// TIA Portal V18 export
FUNCTION_BLOCK "manual_analog"   // FB7, FBD
{ S7_Optimized_Access := 'TRUE' }
VERSION : 0.1
// stored: AutoNumber true, IsIECCheckEnabled false, IsRetainMemResEnabled false, MemoryReserve 100, SetENOAutomatically false, UDAEnableTagReadback false
   VAR_INPUT
      ALLOWED : Bool;
      ALLOWED_ONLY_IN_OVERRIDE : Bool;
      OVERRIDE_NOW : Bool;
      isMultiturn : Bool;
      POS : Real;
      SET_SPEED : Real;
      xFwdOk : Bool;
      xRevOk : Bool;
      clibrated : Bool;
      par_spd_absmax : Real := 1000.0;
      par_dist_absmax : Real := 100.0;
      par_speed_crawl : Real;
      par_dist_crawl : Real;
      par_dist_stop : Real := 10.0;
      par_spd_blind : Real := 500.0;
      par_fwd_limit : Real := 10000.0;
      par_rev_limit : Real := 0.0;
      par_t_acc : Real;
   END_VAR
   VAR_OUTPUT
      SPEED : Real;
      ER_settings : Bool;
      er_ws : WString;
   END_VAR
   VAR
      speed_slowly_accelerated : Real;
      mot_speed_wdir_slowly_accelerated_Instance { S7_SetPoint := 'True'} : "mot_speed_wdir_slowly_accelerated";
   END_VAR
   VAR_TEMP
      speed_calculated : Real;
      speed_calc_abs : Real;
      estop_ok_no_err : Bool;
      blind : Bool;
      set_spd_loc : Real;
   END_VAR
   VAR CONSTANT
      erwsnoer : WString := WSTRING#'no er';
      erws1 : WString := WSTRING#'lim fwd = rev';
      erws2 : WString := WSTRING#'#par_dist_fast 0';
      erws3 : WString := WSTRING#'#par_spd_absmax';
   END_VAR
   VAR_TEMP   // added for the SCL form of the ladder/FBD networks
      _w1 : Bool;
      _w2 : Bool;
   END_VAR
BEGIN

REGION Network 1
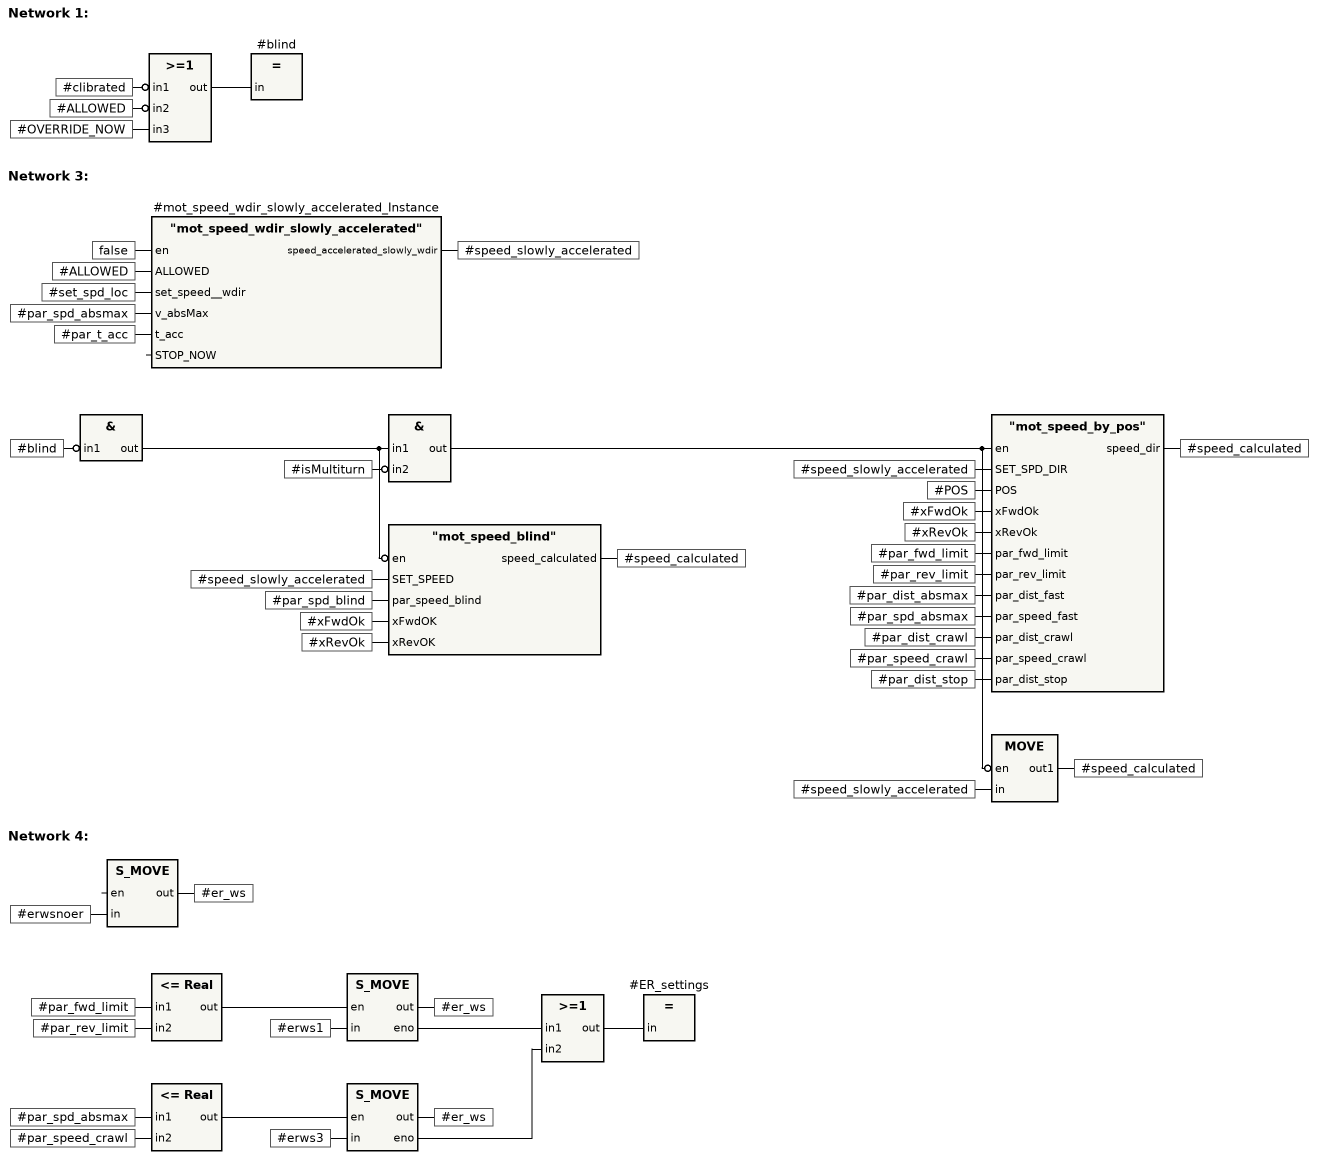
   #blind := NOT #clibrated OR NOT #ALLOWED OR #OVERRIDE_NOW;
END_REGION

REGION Network 2 (SCL)
   #speed_slowly_accelerated := #set_spd_loc := LIMIT(IN:=#SET_SPEED,MN:=-#par_spd_absmax,MX:=#par_spd_absmax);
   //#SET_SPEED*#par_spd_fast
END_REGION

REGION Network 3
   IF false THEN
       #mot_speed_wdir_slowly_accelerated_Instance(ALLOWED := #ALLOWED,   // "mot_speed_wdir_slowly_accelerated"
                               set_speed__wdir := #set_spd_loc,
                               v_absMax := #par_spd_absmax,
                               t_acc := #par_t_acc,
                               speed_accelerated_slowly_wdir => #speed_slowly_accelerated);
   END_IF;
   #_w1 := NOT #blind AND NOT #isMultiturn;
   IF #_w1 THEN
       "mot_speed_by_pos"(SET_SPD_DIR := #speed_slowly_accelerated,
                          POS := #POS,
                          xFwdOk := #xFwdOk,
                          xRevOk := #xRevOk,
                          par_fwd_limit := #par_fwd_limit,
                          par_rev_limit := #par_rev_limit,
                          par_dist_fast := #par_dist_absmax,
                          par_speed_fast := #par_spd_absmax,
                          par_dist_crawl := #par_dist_crawl,
                          par_speed_crawl := #par_speed_crawl,
                          par_dist_stop := #par_dist_stop,
                          speed_dir => #speed_calculated);
   END_IF;
   IF NOT #_w1 THEN #speed_calculated := #speed_slowly_accelerated; END_IF;
   IF NOT (NOT #blind) THEN
       "mot_speed_blind"(SET_SPEED := #speed_slowly_accelerated,
                         par_speed_blind := #par_spd_blind,
                         xFwdOK := #xFwdOk,
                         xRevOK := #xRevOk,
                         speed_calculated => #speed_calculated);
   END_IF;
END_REGION

REGION Network 4
   #er_ws := #erwsnoer;
   #_w1 := #par_fwd_limit <= #par_rev_limit;
   IF #_w1 THEN #er_ws := #erws1; END_IF;
   #_w2 := #par_spd_absmax <= #par_speed_crawl;
   IF #_w2 THEN #er_ws := #erws3; END_IF;
   #ER_settings := #_w1 OR #_w2;
END_REGION

REGION Network 5
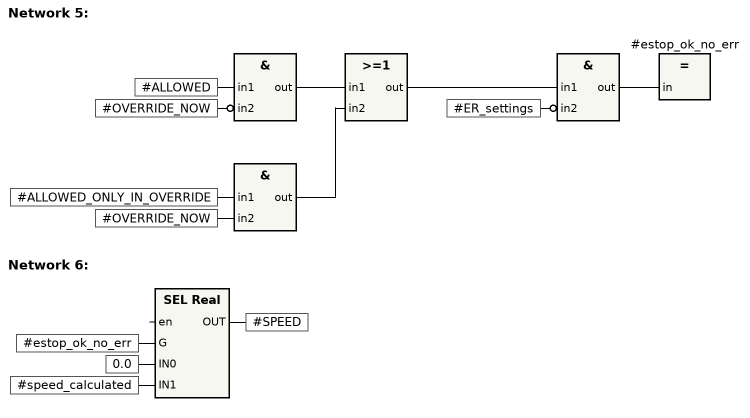
   #estop_ok_no_err := ((#ALLOWED AND NOT #OVERRIDE_NOW) OR (#ALLOWED_ONLY_IN_OVERRIDE AND #OVERRIDE_NOW)) AND NOT #ER_settings;
END_REGION

REGION Network 6
   #SPEED := SEL(G := #estop_ok_no_err, IN0 := 0.0, IN1 := #speed_calculated);
END_REGION
END_FUNCTION_BLOCK
